FUNCTION_BLOCK VCylAdpOL (* Composite Function Block Type *)
  (* Standard: 61499-2 *)
  (* Version 0.0, 06/10/2018, Atmojo, nxtControl GmbH, template *)
  PACKAGE Main;
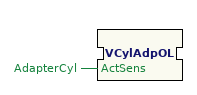
  SOCKETS
    ActSens : AdapterCyl;
  END_SOCKETS
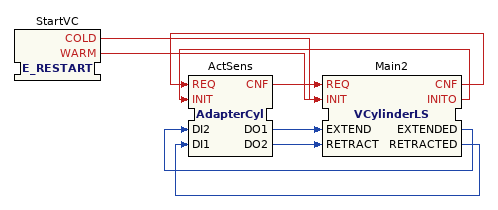
  FBS
    Main2 : VCylinderLS;
    StartVC : E_RESTART;
  END_FBS
  EVENT_CONNECTIONS
    ActSens.CNF TO Main2.REQ;
    StartVC.COLD TO Main2.INIT;
    StartVC.WARM TO Main2.INIT;
    Main2.CNF TO ActSens.REQ;
    Main2.INITO TO ActSens.INIT;
  END_CONNECTIONS
  DATA_CONNECTIONS
    ActSens.DO1 TO Main2.EXTEND;
    ActSens.DO2 TO Main2.RETRACT;
    Main2.EXTENDED TO ActSens.DI2;
    Main2.RETRACTED TO ActSens.DI1;
  END_CONNECTIONS
END_FUNCTION_BLOCK
